Fanuc KAREL source: kd00040.KL

-- PROVISIONAL review KL for V1013-1; original PC SHA256 f50dc470f3220636e6f92f487c0fb60b0a83d1c023b61a78bdd488bd10bade3e
-- Incomplete behavior may be omitted. Consult companion uncertainty JSON. Do not deploy.
PROGRAM KD00040
%NOLOCKGROUP
BEGIN
  -- UNRESOLVED_PC offsets 5-26; opcodes AD,32,22,9B,9B,9C,9C,37,2C
  -- UNRESOLVED_PC offsets 31-35; opcodes 7F
END KD00040
